Omron CX-Programmer project NewProject (CX-Programmer 9.81)

# PLC NewPLC1: CP1L M

## Program NewProgram1 (cyclic task 0)
Local symbols
Contador #0000 NUMBER  ; Contador
M0 5.00 BOOL  ; M0
M1 5.01 BOOL  ; M1
Vf1 100.00 BOOL  ; Variador de Frequência
botao_1 0.00 BOOL  ; Botão 1
botao_2 0.01 BOOL  ; Botão 2
botao_3 0.02 BOOL  ; Botão 3
etapa_0 3.00 BOOL  ; Etapa 0
etapa_1 3.01 BOOL  ; Etapa 1
etapa_2 3.02 BOOL  ; Etapa 2
etapa_3 3.03 BOOL  ; Etapa 3
etapa_4 3.04 BOOL  ; Etapa 4
etapa_5 3.05 BOOL  ; Etapa 5
etapa_6 3.06 BOOL  ; Etapa 6
etapa_7 3.07 BOOL  ; Etapa 7
etapa_8 3.08 BOOL  ; Etapa 8
etapa_9 3.09 BOOL  ; Etapa 9

### Section main

### Section outputs

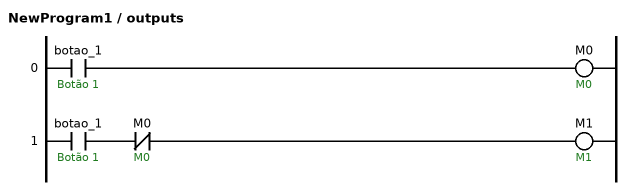
; rung 0
LD botao_1  ; Botão 1
OUT M0  ; M0
; rung 1
LD botao_1  ; Botão 1
ANDNOT M0  ; M0
OUT M1  ; M1
; rung 2
; cells of this rung as drawn
  row 0 col 0: LD M0
  row 0 col 1: wire
  row 0 col 2: wire
  row 0 col 3: wire
  row 0 col 4: wire
  row 0 col 5: wire
  row 0 col 6: CNT #0000 #4
  vertical links (row, left of col): 

### Section timers

### Section END
; rung 0
END(001)